FUNCTION_BLOCK AR_CALIBRATE_3P (* Adapter-based 3-point calibration for joysticks (Min, Mid, Max) *)
  (* Standard: 61499-1 *)
  (* Version 1.1, 2026-09-18, Franz Höpfinger, C_MIN/C_MID/C_MAX von AX-Sockets (mit [C_x.D1]-Flankenwaechter) auf reine EventInputs umgestellt - jeder echte Aufrufer liefert ohnehin ein atomares Event, der D1-Wert war immer hartcodiert TRUE (via AX_BOOL_TO_X) und der Guard filterte nie etwas. Aufrufer muessen jetzt direkt ein Event statt eines AX-Adapters anschliessen. Siehe AR_CALIBRATE_2P_REF fuer die identische Aenderung. *)
  (* Version 1.0, 2026-06-01, Meisterschulen am Ostbahnhof *)
  PACKAGE adapter::Engineering::measurements;
  (* Documentation:
  Formula
   Y = piecewise linear interpolation between stored calibration points Calibration (3-Point)
    - Min (C_MIN): Move joystick to minimum, trigger C_MIN
   X_MIN := X → stores current raw value as Min point
   - Mid (C_MID): Move joystick to center, trigger C_MID
   X_MID := X → stores current raw value as Mid point (center)
   - Max (C_MAX): Move joystick to maximum, trigger C_MAX
   X_MAX := X → stores current raw value as Max point
    Note: Calibration points can be calibrated in any order and repeated individually.
   Output Calculation
    - If X < X_MID: linear interpolation between (X_MIN, MIN_REF) and (X_MID, MID_REF)
   - If X >= X_MID: linear interpolation between (X_MID, MID_REF) and (X_MAX, MAX_REF)
   - Output clipped to MIN_REF..MAX_REF
    Example
   Scenario: Joystick with center drift. Raw range 0..1000, desired output -100..0..100.
    Step | Action | Result | 
   1 | Move joystick to min, trigger C_MIN | X_MIN = 50 (drifted from ideal 0) | 
   2 | Move joystick to center, trigger C_MID | X_MID = 520 (drifted from ideal 500) | 
   3 | Move joystick to max, trigger C_MAX | X_MAX = 980 (drifted from ideal 1000) | 
    Output: Interpolated between MIN_REF=-100, MID_REF=0, MAX_REF=100 with clipping.
  *)
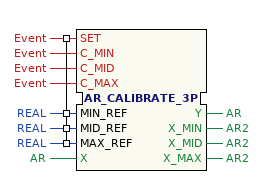
  EVENT_INPUT
    SET WITH MIN_REF, MID_REF, MAX_REF; (* Set Reference Values *)
    C_MIN; (* Calibrate Min Point - atomarer Trigger *)
    C_MID; (* Calibrate Mid Point - atomarer Trigger *)
    C_MAX; (* Calibrate Max Point - atomarer Trigger *)
  END_EVENT
  VAR_INPUT
    MIN_REF : REAL := 0.0; (* Target value for Min *)
    MID_REF : REAL := 50.0; (* Target value for Mid *)
    MAX_REF : REAL := 100.0; (* Target value for Max *)
  END_VAR
  SOCKETS
    X : adapter::types::unidirectional::AR; (* Raw Input *)
  END_SOCKETS
  PLUGS
    Y : adapter::types::unidirectional::AR; (* Calibrated Output *)
    X_MIN : adapter::types::bidirectional::AR2; (* Stored Min Value *)
    X_MID : adapter::types::bidirectional::AR2; (* Stored Mid Value *)
    X_MAX : adapter::types::bidirectional::AR2; (* Stored Max Value *)
  END_PLUGS
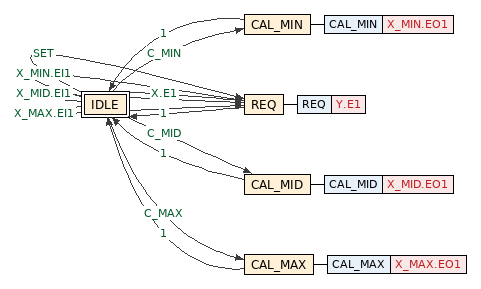
  EC_STATES
    IDLE;
    REQ : REQ -> Y.E1;
    CAL_MIN : CAL_MIN -> X_MIN.EO1;
    CAL_MID : CAL_MID -> X_MID.EO1;
    CAL_MAX : CAL_MAX -> X_MAX.EO1;
  END_STATES
  EC_TRANSITIONS
    IDLE TO REQ := X.E1;
    REQ TO IDLE := 1;
    IDLE TO REQ := SET;
    IDLE TO REQ := X_MIN.EI1;
    IDLE TO REQ := X_MID.EI1;
    IDLE TO REQ := X_MAX.EI1;
    IDLE TO CAL_MIN := C_MIN;
    CAL_MIN TO IDLE := 1;
    IDLE TO CAL_MID := C_MID;
    CAL_MID TO IDLE := 1;
    IDLE TO CAL_MAX := C_MAX;
    CAL_MAX TO IDLE := 1;
  END_TRANSITIONS
  ALGORITHM REQ IN ST:
(* calculate output using stored X_MIN, X_MID, X_MAX from AR2 DI1 ports *)
IF X.D1 < X_MID.DI1 THEN
	IF X_MID.DI1 > X_MIN.DI1 THEN
		Y.D1 := MIN_REF + (X.D1 - X_MIN.DI1) * (MID_REF - MIN_REF) / (X_MID.DI1 - X_MIN.DI1);
	ELSE
		Y.D1 := MIN_REF;
	END_IF;
ELSE
	IF X_MAX.DI1 > X_MID.DI1 THEN
		Y.D1 := MID_REF + (X.D1 - X_MID.DI1) * (MAX_REF - MID_REF) / (X_MAX.DI1 - X_MID.DI1);
	ELSE
		Y.D1 := MID_REF;
	END_IF;
END_IF;

(* clipping *)
IF Y.D1 < MIN_REF THEN
	Y.D1 := MIN_REF;
ELSIF Y.D1 > MAX_REF THEN
	Y.D1 := MAX_REF;
END_IF;
  END_ALGORITHM
  ALGORITHM CAL_MIN IN ST:
X_MIN.DO1 := X.D1;
  END_ALGORITHM
  ALGORITHM CAL_MID IN ST:
X_MID.DO1 := X.D1;
  END_ALGORITHM
  ALGORITHM CAL_MAX IN ST:
X_MAX.DO1 := X.D1;
  END_ALGORITHM
END_FUNCTION_BLOCK
